// TIA Portal V17 export
// export: Created 2023-02-14T02:49:51.418011Z, ExportSetting WithDefaults, DisplayName Totally Integrated Automation Portal, DisplayVersion V17, DisplayName TIA Portal Openness, DisplayVersion V17, DisplayName TIA Portal Teamcenter Gateway, DisplayVersion V17, DisplayName TIA Portal Version Control Interface, DisplayVersion V17, DisplayName SINAMICS Startdrive Advanced, DisplayVersion V17, DisplayName SINAMICS Startdrive G130, G150, S120, S150, SINAMICS MV, S210, DisplayVersion V17, DisplayName SINAMICS Startdrive G110M, G120, G120C, G120D, G120P, G115D, DisplayVersion V17, DisplayName STEP 7 Professional, DisplayVersion V17, DisplayName STEP 7 Safety, DisplayVersion V17, DisplayName WinCC Professional, DisplayVersion V17
FUNCTION_BLOCK "Rework"   // FB32, LAD
{ S7_Optimized_Access := 'FALSE' }
VERSION : 0.1
// stored: AutoNumber false, IsIECCheckEnabled false, SetENOAutomatically false, UDAEnableTagReadback false
   VAR_INPUT
      Level_Bypass_JBT : Bool;
      Single_CIP_Cmd : Bool;
      IN_FBAV_Load : Bool;
      IN_FBAV_Transfer : Bool;
      IN_FBP_Transfer : Bool;
      IN_FBP_Transfer_Speed : Real;
      IN_FBP_CIP : Bool;
      IN_FBAV_CIP_Sup : Bool;
      IN_FBAV_CIP_Tank : Bool;
      IN_FBAV_CIP_Line : Bool;
      IN_LT01 : Real;
      IN_FS : Bool;
      CIP_Req_OK : Bool;
      CIP_ON_Progress : Bool;
      CIP_Supply_ON : Bool;
      CIP_Complete : Bool;
      CIPPulse : Bool;
      Filler_Product_Req : Bool;
      Filler_CIP_Req : Bool;
      Loading_Busy : Bool;
      Transfer_Busy : Bool;
   END_VAR
   VAR_OUTPUT
      Out_AV_Load : Bool;
      Out_AV_Transfer : Bool;
      Out_P_Transfer : Bool;
      Out_P_TF_Speed : Real;
      Out_P_CIP : Bool;
      Out_P_Circ : Bool;
      Out_P_Circ_Speed : Real;
      Out_AV_CIP_Line : Bool;
      Out_AV_CIP_Tank : Bool;
      Out_AV_CIP_Filling : Bool;
      CIP_Tank_Req : Bool;
      CIP_Line_Req : Bool;
      CIP_LineOK : Bool;
   END_VAR
   VAR DB_SPECIFIC
      Cmd : Struct
         Inload_Select_Tank : Bool;
         Inload : Bool;   // Start Loading
         Tank_CIP_Req : Bool;
         Line_CIP_Req : Bool;
         Tank_Filling_CIP_Req : Bool;
         CIP_Filling_En : Bool;
         CIP_Line_Req_OK : Bool;
         CIP_Supply_ON : Bool;
         CIP_ON_Progress : Bool;
         Transfer : Bool;   // Water Flushing
         RaadyForTF : Bool;   // Tank Ready for Blending
         Flush_Select : Byte;
         Drain_In : Bool;
         Drain_Transfer : Bool;
         Circulation_CMD_ON : Bool := true;
         free : Bool;
         free_1 : Bool;
         free_2 : Bool;
         free_3 : Bool;
      END_STRUCT;
      Param : Struct
         SP_Level_LL : Real := 10.0;
         SP_Level_ML : Real := 80.0;
         SP_Level_HL : Real := 100.0;
         SupplyPump_SP_Speed : Real := 80.0;
         L_Hi_Lim : Real := 100.0;
         L_Lo_Lim : Real := 0.0;
         L_Hys : Real := 5.0;
         FlushingTime : DInt := 10000;
         CIP_Trf_SP_Speed : Real := 80.0;
         CIP_Ret_ON_SP : Real := 10.0;
         CIP_Ret_OFF_SP : Real;
         Transfer_P_Speed : Real := 60.0;
         Drain_Inload_SP : DInt := 10;
         Drain_Transfer_SP : DInt := 10;
         "Circulation Level" : Real := 50.0;
         free : DInt;
         free_1 : DInt;
         free_2 : Real;
         free_3 : Real;
         free_4 : Real;
      END_STRUCT;
      State : Struct   // Tank in loading state
         Tank_inloading : Bool;
         Tank_inCIP : Bool;
         Tank_Filling_inCIP : Bool;
         Line_inCIP : Bool;
         FIlling_inCIP : Bool;
         Flushing : Bool;
         Tank_LL : Bool;
         Tank_ML : Bool;
         Tank_HL : Bool;
         Inload_Enable : Bool;
         Tank_CIP_Enable : Bool;
         Line_CIP_Enable : Bool;
         Tank_Filling_CIP_Enable : Bool;
         Flushing_Enable : Bool;
         Flush_selected : Byte;
         CIP_Request_OK : Bool;
         CIP_ReturnON : Bool;
         Ready_For_Transfer_EN : Bool;   // Tank Ready for Transfer to Blending
         Ready_For_Transfer : Bool;   // Tank Ready for Transfer to Blending
         HWT_Status : Int;
         Transfer_to_Filling : Bool;
         "Line_AV4&AV5" : Bool;
         "Line_AV1&AV2" : Bool;
         "Line_AV7&AV8" : Bool;
         "Line_AV10&AV11" : Bool;
         "Line_AV5&AV6" : Bool;
         CIP_Line1_ON : Bool;
         CIP_Line2_ON : Bool;
         CIP_Line3_ON : Bool;
         CIP_Line4_ON : Bool;
         Drain_Inload : Bool;
         Drain_Transfer : Bool;
         "Circulation Enable" : Bool;
         Circulation_ON : Bool;
         Tank_Circulation : Bool;
         HighLevel_Coll_Tank : Bool;
         Alarm_Prod : Bool;
         free_2 : Bool;
         free_3 : Bool;
      END_STRUCT;
      alwaysON : Bool;
      L_Hys_Abs : Real;
      Hys_Level_HL : Real;
      Hys_Level_ML : Real;
      Hys_Level_LL : Real;
      Hys_Level_Circ : Real;
      Drain_Inload_MSec : DInt;
      Drain_Inload_Count : IEC_DCOUNTER;
      Drain_Inload_Act { S7_SetPoint := 'True'} : DInt;
      Drain_Transfer_MSec : DInt;
      Drain_Transfer_Count : IEC_DCOUNTER;
      Drain_Transfer_Act : DInt;
      r : Struct
         PosE1 : Bool;
         PosE2 : Bool;
         PosE3 : Bool;
         PosE4 : Bool;
         PosE5 : Bool;
         PosE6 : Bool;
         PosE7 : Bool;
         PosE8 : Bool;
         PosE9 : Bool;
         PosE10 : Bool;
         PosE11 : Bool;
         PosE12 : Bool;
         PosE13 : Bool;
         PosE14 : Bool;
         PosE15 : Bool;
         PosE16 : Bool;
         PosE17 : Bool;
         PosE18 : Bool;
         PosE19 : Bool;
         PosE20 : Bool;
         PosE21 : Bool;
         PosE22 : Bool;
         PosE23 : Bool;
         PosE24 : Bool;
         PosE25 : Bool;
         PosE26 : Bool;
         PosE27 : Bool;
         PosE28 : Bool;
         PosE29 : Bool;
         PosE30 : Bool;
         PosE31 : Bool;
         PosE32 : Bool;
      END_STRUCT;
      Actuator : Struct
         AV_Outlet : Bool;
         AV_Load : Bool;
         AV_Transfer : Bool;
         CIP_Line_Pump : Bool;
         CIP_Tank_Pump : Bool;
         TransferPump : Bool;
         FlushPump : Bool;
         CV_Steam : Bool;
         Pump : Bool;
      END_STRUCT;
      SPumpTim { S7_SetPoint := 'True'} : TON_TIME;
      SAV_CIPLine { S7_SetPoint := 'True'} : TON_TIME;
      SAV_CIPTANK { S7_SetPoint := 'True'} : TON_TIME;
      SAV_CIPFILLING { S7_SetPoint := 'True'} : TON_TIME;
      AVinloadTim { S7_SetPoint := 'True'} : TON_TIME;
      AVOutletTim { S7_SetPoint := 'True'} : TON_TIME;
      Drain_In_Tim { S7_SetPoint := 'True'} : TON_TIME;
      Drain_Out_Tim { S7_SetPoint := 'True'} : TON_TIME;
      "Pump Off Tim" { S7_SetPoint := 'True'} : TON_TIME;
      "Loading_Busy Tim" { S7_SetPoint := 'True'} : TON_TIME;
   END_VAR
   VAR_TEMP   // added for the SCL form of the ladder/FBD networks
      _w1 : Bool;
      _w2 : Bool;
   END_VAR
BEGIN

REGION Network 1: Always ON
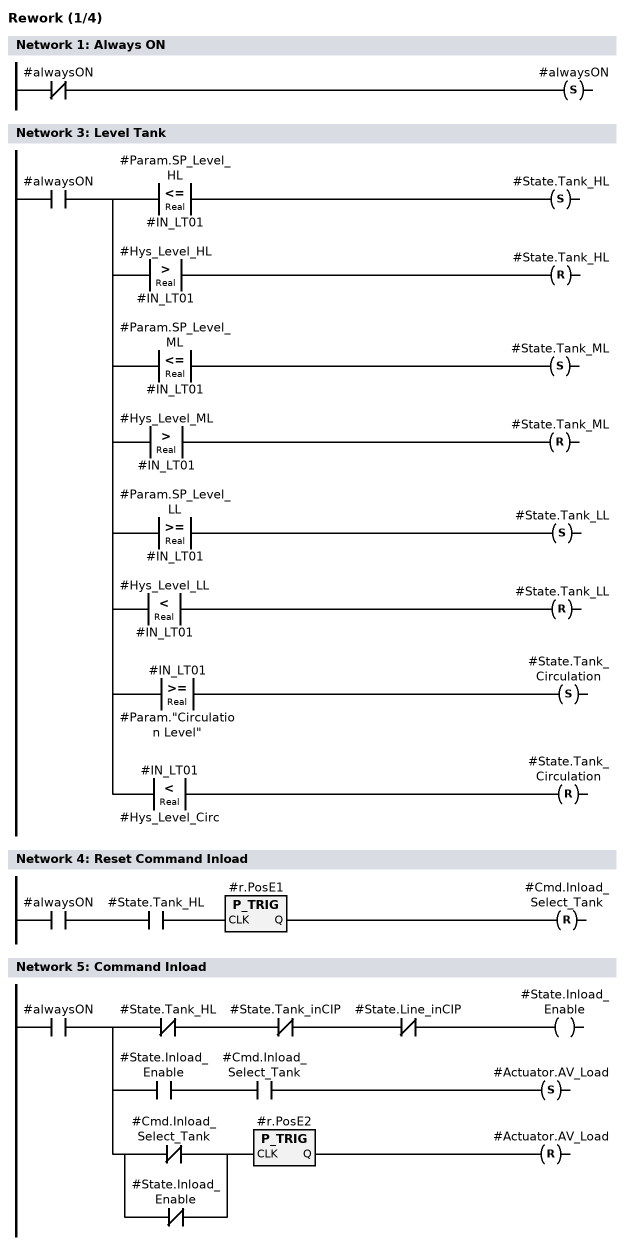
   RUNG wire#powerrail
      I_Contact( #alwaysON )
      S_Coil( #alwaysON )
   END_RUNG
   // the same network as SCL:
   IF NOT #alwaysON THEN #alwaysON := TRUE; END_IF;
END_REGION

NETWORK
TITLE = Hys Calculation
//Level Hys Absolute
      L     #Param.L_Hi_Lim;
      L     #Param.L_Lo_Lim;
      -R;
      L     100.0;
      /R;
      L     #Param.L_Hys;
      *R;
      T     #L_Hys_Abs;
//Tank High Level
      L     #Param.SP_Level_HL;
      L     #L_Hys_Abs;
      -R;
      T     #Hys_Level_HL;
//Tank Mid Level
      L     #Param.SP_Level_ML;
      L     #L_Hys_Abs;
      -R;
      T     #Hys_Level_ML;
//Tank Low Level
      L     #Param.SP_Level_LL;
      L     #L_Hys_Abs;
      +R;
      T     #Hys_Level_LL;
//Level Circulation
      L     #Param."Circulation Level";
      L     #L_Hys_Abs;
      -R;
      T     #Hys_Level_Circ;



REGION Network 3: Level Tank
   RUNG wire#powerrail
      Contact( #alwaysON )
      wire#w1
      { S7_Templates := "SrcType := Real" } LE_Contact(in1 := #Param.SP_Level_HL, in2 := #IN_LT01)
      S_Coil( #State.Tank_HL )
   END_RUNG
   RUNG wire#w1
      { S7_Templates := "SrcType := Real" } GT_Contact(in1 := #Hys_Level_HL, in2 := #IN_LT01)
      R_Coil( #State.Tank_HL )
   END_RUNG
   RUNG wire#w1
      { S7_Templates := "SrcType := Real" } LE_Contact(in1 := #Param.SP_Level_ML, in2 := #IN_LT01)
      S_Coil( #State.Tank_ML )
   END_RUNG
   RUNG wire#w1
      { S7_Templates := "SrcType := Real" } GT_Contact(in1 := #Hys_Level_ML, in2 := #IN_LT01)
      R_Coil( #State.Tank_ML )
   END_RUNG
   RUNG wire#w1
      { S7_Templates := "SrcType := Real" } GE_Contact(in1 := #Param.SP_Level_LL, in2 := #IN_LT01)
      S_Coil( #State.Tank_LL )
   END_RUNG
   RUNG wire#w1
      { S7_Templates := "SrcType := Real" } LT_Contact(in1 := #Hys_Level_LL, in2 := #IN_LT01)
      R_Coil( #State.Tank_LL )
   END_RUNG
   RUNG wire#w1
      { S7_Templates := "SrcType := Real" } GE_Contact(in1 := #IN_LT01, in2 := #Param."Circulation Level")
      S_Coil( #State.Tank_Circulation )
   END_RUNG
   RUNG wire#w1
      { S7_Templates := "SrcType := Real" } LT_Contact(in1 := #IN_LT01, in2 := #Hys_Level_Circ)
      R_Coil( #State.Tank_Circulation )
   END_RUNG
   // the same network as SCL:
   IF #alwaysON AND (#Param.SP_Level_HL <= #IN_LT01) THEN #State.Tank_HL := TRUE; END_IF;
   IF #alwaysON AND (#Hys_Level_HL > #IN_LT01) THEN #State.Tank_HL := FALSE; END_IF;
   IF #alwaysON AND (#Param.SP_Level_ML <= #IN_LT01) THEN #State.Tank_ML := TRUE; END_IF;
   IF #alwaysON AND (#Hys_Level_ML > #IN_LT01) THEN #State.Tank_ML := FALSE; END_IF;
   IF #alwaysON AND (#Param.SP_Level_LL >= #IN_LT01) THEN #State.Tank_LL := TRUE; END_IF;
   IF #alwaysON AND (#Hys_Level_LL < #IN_LT01) THEN #State.Tank_LL := FALSE; END_IF;
   IF #alwaysON AND (#IN_LT01 >= #Param."Circulation Level") THEN #State.Tank_Circulation := TRUE; END_IF;
   IF #alwaysON AND (#IN_LT01 < #Hys_Level_Circ) THEN #State.Tank_Circulation := FALSE; END_IF;
END_REGION

REGION Network 4: Reset Command Inload
   RUNG wire#powerrail
      Contact( #alwaysON )
      Contact( #State.Tank_HL )
      P_Trig( #r.PosE1 )
      R_Coil( #Cmd.Inload_Select_Tank )
   END_RUNG
   // the same network as SCL:
   #_w1 := #alwaysON AND #State.Tank_HL;
   #_w2 := #_w1 AND NOT #r.PosE1;   // rising edge
   #r.PosE1 := #_w1;
   IF #_w2 THEN #Cmd.Inload_Select_Tank := FALSE; END_IF;
END_REGION

REGION Network 5: Command Inload
   RUNG wire#powerrail
      Contact( #alwaysON )
      wire#w1
      I_Contact( #State.Tank_HL )
      I_Contact( #State.Tank_inCIP )
      I_Contact( #State.Line_inCIP )
      Coil( #State.Inload_Enable )
   END_RUNG
   RUNG wire#w1
      Contact( #State.Inload_Enable )
      Contact( #Cmd.Inload_Select_Tank )
      S_Coil( #Actuator.AV_Load )
   END_RUNG
   RUNG wire#w1
      I_Contact( #Cmd.Inload_Select_Tank )
      wire#w2
      P_Trig( #r.PosE2 )
      R_Coil( #Actuator.AV_Load )
   END_RUNG
   RUNG wire#w1
      I_Contact( #State.Inload_Enable )
   END_RUNG wire#w2
   // the same network as SCL:
   #State.Inload_Enable := #alwaysON AND NOT #State.Tank_HL AND NOT #State.Tank_inCIP AND NOT #State.Line_inCIP;
   IF #alwaysON AND #State.Inload_Enable AND #Cmd.Inload_Select_Tank THEN #Actuator.AV_Load := TRUE; END_IF;
   #_w1 := #alwaysON AND (NOT #Cmd.Inload_Select_Tank OR NOT #State.Inload_Enable);
   #_w2 := #_w1 AND NOT #r.PosE2;   // rising edge
   #r.PosE2 := #_w1;
   IF #_w2 THEN #Actuator.AV_Load := FALSE; END_IF;
END_REGION

REGION Network 6: Command Transfer to Filling
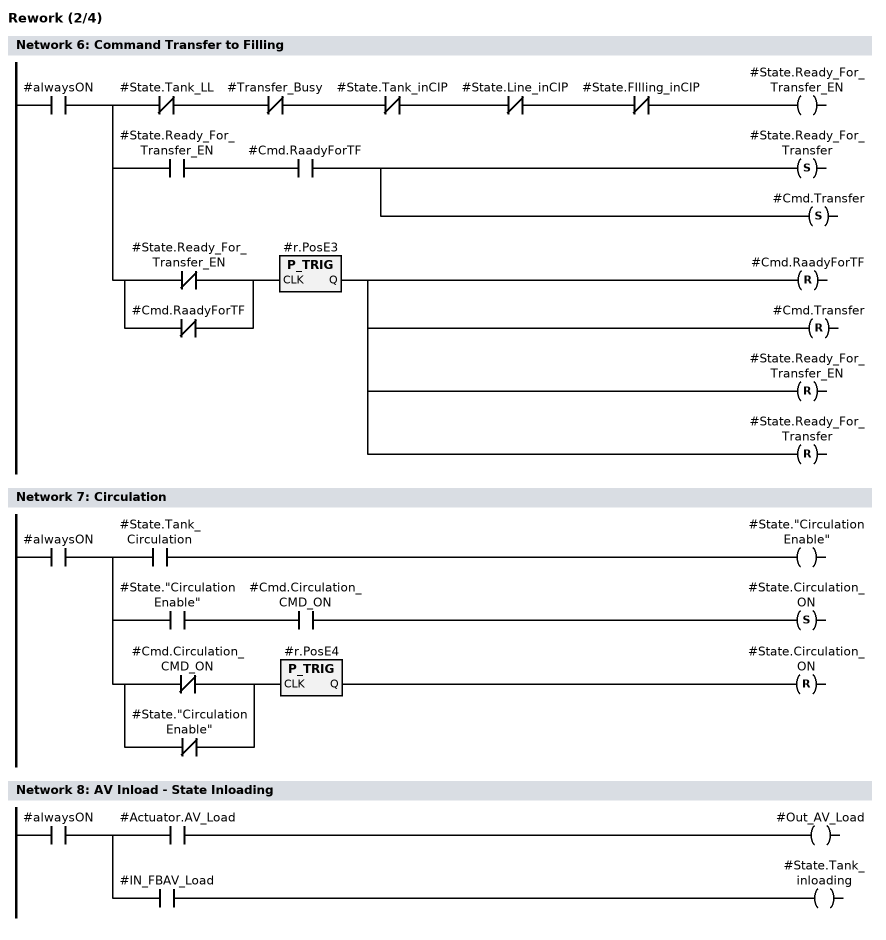
   RUNG wire#powerrail
      Contact( #alwaysON )
      wire#w1
      I_Contact( #State.Tank_LL )
      I_Contact( #Transfer_Busy )
      I_Contact( #State.Tank_inCIP )
      I_Contact( #State.Line_inCIP )
      I_Contact( #State.FIlling_inCIP )
      Coil( #State.Ready_For_Transfer_EN )
   END_RUNG
   RUNG wire#w1
      Contact( #State.Ready_For_Transfer_EN )
      Contact( #Cmd.RaadyForTF )
      wire#w2
      S_Coil( #State.Ready_For_Transfer )
   END_RUNG
   RUNG wire#w2
      S_Coil( #Cmd.Transfer )
   END_RUNG
   RUNG wire#w1
      I_Contact( #State.Ready_For_Transfer_EN )
      wire#w3
      P_Trig( #r.PosE3 )
      wire#w4
      R_Coil( #Cmd.RaadyForTF )
   END_RUNG
   RUNG wire#w1
      I_Contact( #Cmd.RaadyForTF )
   END_RUNG wire#w3
   RUNG wire#w4
      R_Coil( #Cmd.Transfer )
   END_RUNG
   RUNG wire#w4
      R_Coil( #State.Ready_For_Transfer_EN )
   END_RUNG
   RUNG wire#w4
      R_Coil( #State.Ready_For_Transfer )
   END_RUNG
   // the same network as SCL:
   #State.Ready_For_Transfer_EN := #alwaysON AND NOT #State.Tank_LL AND NOT #Transfer_Busy AND NOT #State.Tank_inCIP AND NOT #State.Line_inCIP AND NOT #State.FIlling_inCIP;
   IF #alwaysON AND #State.Ready_For_Transfer_EN AND #Cmd.RaadyForTF THEN
       #State.Ready_For_Transfer := TRUE;
       #Cmd.Transfer := TRUE;
   END_IF;
   #_w1 := #alwaysON AND (NOT #State.Ready_For_Transfer_EN OR NOT #Cmd.RaadyForTF);
   #_w2 := #_w1 AND NOT #r.PosE3;   // rising edge
   #r.PosE3 := #_w1;
   IF #_w2 THEN
       #Cmd.RaadyForTF := FALSE;
       #Cmd.Transfer := FALSE;
       #State.Ready_For_Transfer_EN := FALSE;
       #State.Ready_For_Transfer := FALSE;
   END_IF;
END_REGION

REGION Network 7: Circulation
   RUNG wire#powerrail
      Contact( #alwaysON )
      wire#w1
      Contact( #State.Tank_Circulation )
      Coil( #State."Circulation Enable" )
   END_RUNG
   RUNG wire#w1
      Contact( #State."Circulation Enable" )
      Contact( #Cmd.Circulation_CMD_ON )
      S_Coil( #State.Circulation_ON )
   END_RUNG
   RUNG wire#w1
      I_Contact( #Cmd.Circulation_CMD_ON )
      wire#w2
      P_Trig( #r.PosE4 )
      R_Coil( #State.Circulation_ON )
   END_RUNG
   RUNG wire#w1
      I_Contact( #State."Circulation Enable" )
   END_RUNG wire#w2
   // the same network as SCL:
   #State."Circulation Enable" := #alwaysON AND #State.Tank_Circulation;
   IF #alwaysON AND #State."Circulation Enable" AND #Cmd.Circulation_CMD_ON THEN
       #State.Circulation_ON := TRUE;
   END_IF;
   #_w1 := #alwaysON AND (NOT #Cmd.Circulation_CMD_ON OR NOT #State."Circulation Enable");
   #_w2 := #_w1 AND NOT #r.PosE4;   // rising edge
   #r.PosE4 := #_w1;
   IF #_w2 THEN #State.Circulation_ON := FALSE; END_IF;
END_REGION

REGION Network 8: AV Inload - State Inloading
   RUNG wire#powerrail
      Contact( #alwaysON )
      wire#w1
      Contact( #Actuator.AV_Load )
      Coil( #Out_AV_Load )
   END_RUNG
   RUNG wire#w1
      Contact( #IN_FBAV_Load )
      Coil( #State.Tank_inloading )
   END_RUNG
   // the same network as SCL:
   #Out_AV_Load := #alwaysON AND #Actuator.AV_Load;
   #State.Tank_inloading := #alwaysON AND #IN_FBAV_Load;
END_REGION

REGION Network 9: AV Transfer / Output
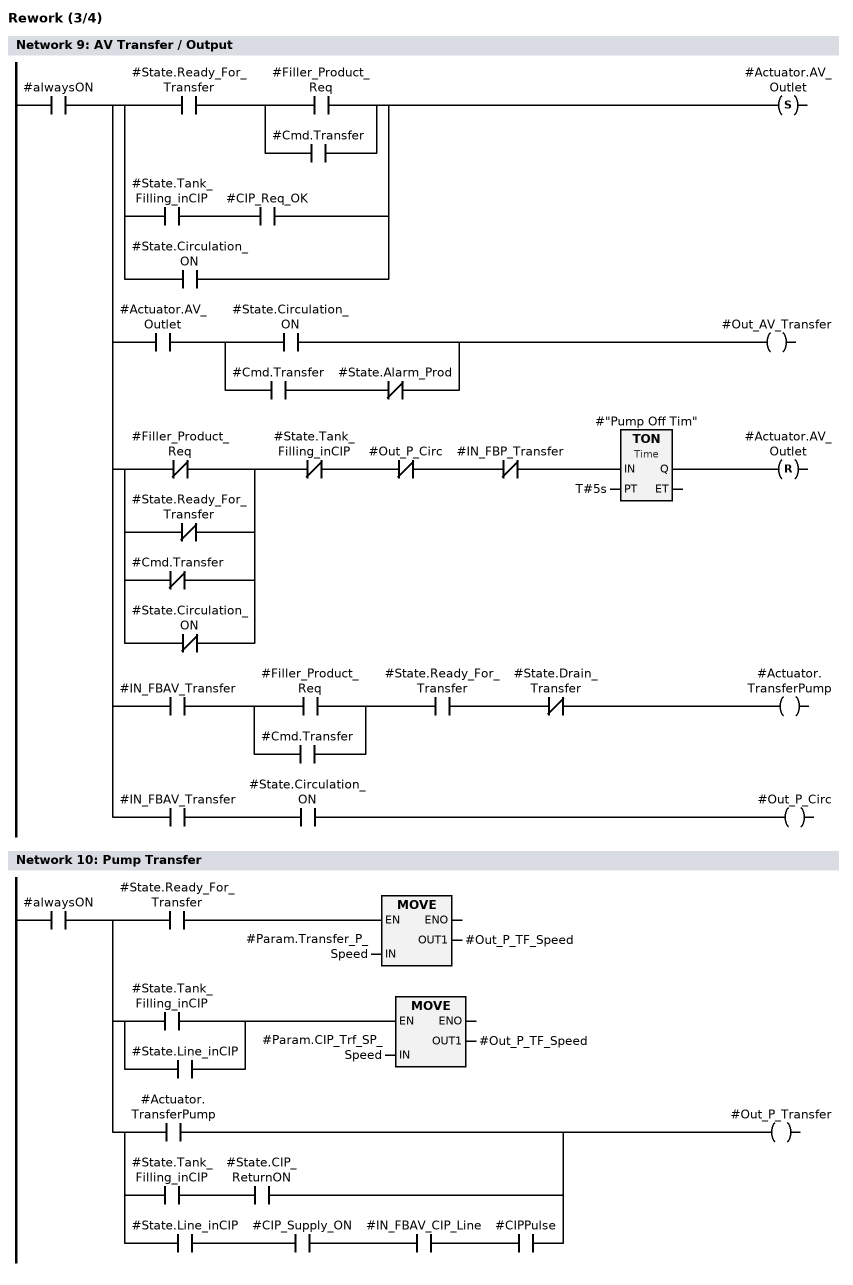
   RUNG wire#powerrail
      Contact( #alwaysON )
      wire#w1
      Contact( #State.Ready_For_Transfer )
      wire#w2
      Contact( #Filler_Product_Req )
      wire#w3
      S_Coil( #Actuator.AV_Outlet )
   END_RUNG
   RUNG wire#w2
      Contact( #Cmd.Transfer )
   END_RUNG wire#w3
   RUNG wire#w1
      Contact( #State.Tank_Filling_inCIP )
      Contact( #CIP_Req_OK )
   END_RUNG wire#w3
   RUNG wire#w1
      Contact( #State.Circulation_ON )
   END_RUNG wire#w3
   RUNG wire#w1
      Contact( #Actuator.AV_Outlet )
      wire#w4
      Contact( #State.Circulation_ON )
      wire#w5
      Coil( #Out_AV_Transfer )
   END_RUNG
   RUNG wire#w4
      Contact( #Cmd.Transfer )
      I_Contact( #State.Alarm_Prod )
   END_RUNG wire#w5
   RUNG wire#w1
      I_Contact( #Filler_Product_Req )
      wire#w6
      I_Contact( #State.Tank_Filling_inCIP )
      I_Contact( #Out_P_Circ )
      I_Contact( #IN_FBP_Transfer )
      { S7_Templates := "time_type := Time" } #"Pump Off Tim".TON(pt := T#5s, et =>)
      R_Coil( #Actuator.AV_Outlet )
   END_RUNG
   RUNG wire#w1
      I_Contact( #State.Ready_For_Transfer )
   END_RUNG wire#w6
   RUNG wire#w1
      I_Contact( #Cmd.Transfer )
   END_RUNG wire#w6
   RUNG wire#w1
      I_Contact( #State.Circulation_ON )
   END_RUNG wire#w6
   RUNG wire#w1
      Contact( #IN_FBAV_Transfer )
      wire#w7
      Contact( #Filler_Product_Req )
      wire#w8
      Contact( #State.Ready_For_Transfer )
      I_Contact( #State.Drain_Transfer )
      Coil( #Actuator.TransferPump )
   END_RUNG
   RUNG wire#w7
      Contact( #Cmd.Transfer )
   END_RUNG wire#w8
   RUNG wire#w1
      Contact( #IN_FBAV_Transfer )
      Contact( #State.Circulation_ON )
      Coil( #Out_P_Circ )
   END_RUNG
   // the same network as SCL:
   IF #alwaysON AND ((#State.Ready_For_Transfer AND (#Filler_Product_Req OR #Cmd.Transfer)) OR (#State.Tank_Filling_inCIP AND #CIP_Req_OK) OR #State.Circulation_ON) THEN
       #Actuator.AV_Outlet := TRUE;
   END_IF;
   #Out_AV_Transfer := #alwaysON AND #Actuator.AV_Outlet AND (#State.Circulation_ON OR (#Cmd.Transfer AND NOT #State.Alarm_Prod));
   #"Pump Off Tim"(IN := #alwaysON AND (NOT #Filler_Product_Req OR NOT #State.Ready_For_Transfer OR NOT #Cmd.Transfer OR NOT #State.Circulation_ON) AND NOT #State.Tank_Filling_inCIP AND NOT #Out_P_Circ AND NOT #IN_FBP_Transfer,   // TON
                   PT := T#5s);
   IF #"Pump Off Tim".Q THEN #Actuator.AV_Outlet := FALSE; END_IF;
   #Actuator.TransferPump := #alwaysON AND #IN_FBAV_Transfer AND (#Filler_Product_Req OR #Cmd.Transfer) AND #State.Ready_For_Transfer AND NOT #State.Drain_Transfer;
   #Out_P_Circ := #alwaysON AND #IN_FBAV_Transfer AND #State.Circulation_ON;
END_REGION

REGION Network 10: Pump Transfer
   RUNG wire#powerrail
      Contact( #alwaysON )
      wire#w1
      Contact( #State.Ready_For_Transfer )
      Move(in := #Param.Transfer_P_Speed, out1 => #Out_P_TF_Speed)
   END_RUNG
   RUNG wire#w1
      Contact( #State.Tank_Filling_inCIP )
      wire#w2
      Move(in := #Param.CIP_Trf_SP_Speed, out1 => #Out_P_TF_Speed)
   END_RUNG
   RUNG wire#w1
      Contact( #State.Line_inCIP )
   END_RUNG wire#w2
   RUNG wire#w1
      Contact( #Actuator.TransferPump )
      wire#w3
      Coil( #Out_P_Transfer )
   END_RUNG
   RUNG wire#w1
      Contact( #State.Tank_Filling_inCIP )
      Contact( #State.CIP_ReturnON )
   END_RUNG wire#w3
   RUNG wire#w1
      Contact( #State.Line_inCIP )
      Contact( #CIP_Supply_ON )
      Contact( #IN_FBAV_CIP_Line )
      Contact( #CIPPulse )
   END_RUNG wire#w3
   // the same network as SCL:
   IF #alwaysON AND #State.Ready_For_Transfer THEN #Out_P_TF_Speed := #Param.Transfer_P_Speed; END_IF;
   IF #alwaysON AND (#State.Tank_Filling_inCIP OR #State.Line_inCIP) THEN
       #Out_P_TF_Speed := #Param.CIP_Trf_SP_Speed;
   END_IF;
   #Out_P_Transfer := #alwaysON AND (#Actuator.TransferPump OR (#State.Tank_Filling_inCIP AND #State.CIP_ReturnON) OR (#State.Line_inCIP AND #CIP_Supply_ON AND #IN_FBAV_CIP_Line AND #CIPPulse));
END_REGION

REGION Network 11: State Transfer to FIlling
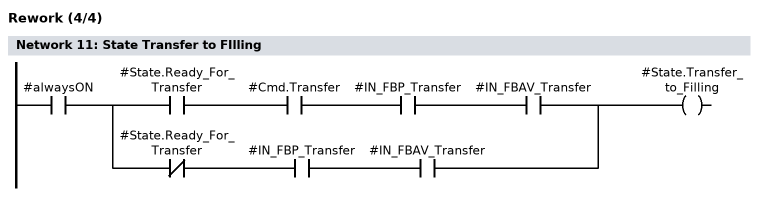
   RUNG wire#powerrail
      Contact( #alwaysON )
      wire#w1
      Contact( #State.Ready_For_Transfer )
      Contact( #Cmd.Transfer )
      Contact( #IN_FBP_Transfer )
      Contact( #IN_FBAV_Transfer )
      wire#w2
      Coil( #State.Transfer_to_Filling )
   END_RUNG
   RUNG wire#w1
      I_Contact( #State.Ready_For_Transfer )
      Contact( #IN_FBP_Transfer )
      Contact( #IN_FBAV_Transfer )
   END_RUNG wire#w2
   // the same network as SCL:
   #State.Transfer_to_Filling := #alwaysON AND ((#State.Ready_For_Transfer AND #Cmd.Transfer AND #IN_FBP_Transfer AND #IN_FBAV_Transfer) OR (NOT #State.Ready_For_Transfer AND #IN_FBP_Transfer AND #IN_FBAV_Transfer));
END_REGION
END_FUNCTION_BLOCK
